// TIA Portal V18 export
DATA_BLOCK "DB_FB_Storer_0"   // DB14
VERSION : 0.1
// stored: AutoNumber true, DBAccessibleFromOPCUA true, DBAccessibleFromWebserver true, InstanceOfName FB_Storer, InstanceOfType FB
"FB_Storer"
   // VAR_INPUT
   //    in_manual : Bool;
   //    in_manualHorizontalPoint : Real;
   //    in_manualVeticalPoint : Real;
   // END_VAR
   // VAR_OUTPUT
   //    out_succes : Bool;
   //    out_ocupied : Bool;
   // END_VAR
   // VAR
   //    horizontal_point : Int;
   //    vertical_point : Int;
   //    hortizontal_converted { ExternalAccessible := 'False'; ExternalVisible := 'False'; ExternalWritable := 'False'} : Real;
   //    vertical_converted { ExternalAccessible := 'False'; ExternalVisible := 'False'; ExternalWritable := 'False'} : Real;
   //    Storer : Array[0..4] of "udt_StoreRow";
   //    Storer_box_type { S7_SetPoint := 'True'} : Array[0..4] of "udt_StoreRowBoxType";
   // END_VAR
BEGIN
END_DATA_BLOCK
